// TIA Portal V21 export
FUNCTION "Motore_PompaRilancioTorre" : Void   // FC134, LAD
{ S7_Optimized_Access := 'TRUE' }
// stored: SetENOAutomatically false
   VAR_TEMP
      AutoPos : Bool;
      AutoNeg : Bool;
   END_VAR
BEGIN

REGION Network 1: Comando positivo in automatico
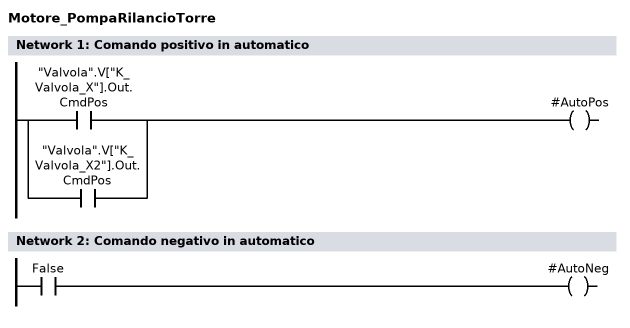
   RUNG wire#powerrail
      Contact( "Valvola".V["K_Valvola_X"].Out.CmdPos )
      wire#w1
      Coil( #AutoPos )
   END_RUNG
   RUNG wire#powerrail
      Contact( "Valvola".V["K_Valvola_X2"].Out.CmdPos )
   END_RUNG wire#w1
   // the same network as SCL:
   #AutoPos := "Valvola".V["K_Valvola_X"].Out.CmdPos OR "Valvola".V["K_Valvola_X2"].Out.CmdPos;
END_REGION

REGION Network 2: Comando negativo in automatico
   RUNG wire#powerrail
      Contact( False )
      Coil( #AutoNeg )
   END_RUNG
   // the same network as SCL:
   #AutoNeg := False;
END_REGION

REGION Network 3 (SCL)
   REGION PompaRilancioTorre
       REGION Ingressi
           "Motore".M[K_Motore_PompaRilancioTorre].In.FbDigitali.FaultInverter := NOT "PompaRilancioTorre_Ready";
           "Motore".M[K_Motore_PompaRilancioTorre].In.FbDigitali.FeedbackMarcia := "PompaRilancioTorre_Marcia";
           "Motore".M[K_Motore_PompaRilancioTorre].In.CmdPosRich := #AutoPos;
           "Motore".M[K_Motore_PompaRilancioTorre].In.CmdNegRich := #AutoNeg;
       END_REGION ;
       REGION
           "GestMotore"(K_Motore := "K_Motore_PompaRilancioTorre",
                        K_TipoMotore := "K_TipoMotore_InverterKEB",
                        K_Zona := "K_Zona_Sterilizzatore");
       END_REGION ;
       REGION Uscite 
           "PompaRilancioTorre_ComandoMarcia" := "Motore".M[K_Motore_PompaRilancioTorre].Out.CmdPosMotore;
           "PompaRilancioTorre_Velocità" := DINT_TO_WORD("Motore".M[K_Motore_PompaRilancioTorre].Out.Paw);
       END_REGION ;
   END_REGION ;
END_REGION
END_FUNCTION
